PROGRAM P_Demo_GetCoreTemperature
VAR
    fbCBM            : TC_CoreBoostMonitor; // TC_CoreBoostMonitor 实例
    hrResult         : HRESULT; // 方法返回的 HRESULT
    out_nCurrentTemp : UDINT; // 方法 REFERENCE TO nCurrentTemp 出参
    out_nMaxTemp     : UDINT; // 方法 REFERENCE TO nMaxTemp 出参
    out_nTempLimit   : UDINT; // 方法 REFERENCE TO nTempLimit 出参
END_VAR

// ============================================================
// Tc2_Utilities.TC_CoreBoostMonitor.GetCoreTemperature 演示程序（METHOD）
// ============================================================
// 注意：必须 Intel Core i 11 代+ 且 TwinCAT Core Boost 已启用
// 验证步骤：
//   1. 引用 Tc2_Utilities
//   2. 编译 + 登录
//   3. 在 Real-time Settings 启用 Core Boost
//   4. 在线监视 hrResult 与 out_* 出参
// ============================================================

hrResult := fbCBM.GetCoreTemperature(out_nCurrentTemp, out_nMaxTemp, out_nTempLimit);

END_PROGRAM

(* stored: Version 1.1.0.1, ProductVersion 3.1.4024.5
   POU P_Demo_GetCoreTemperature: Id {5376785e-a9a5-5675-bbb4-69b42184b678}, SpecialFunc None *)
